FUNCTION_BLOCK  CycleHandleFB 
VAR_IN_OUT

END_VAR

VAR_INPUT
	//pFlowID: 			POINTER TO DINT :=ADR(DummyFlowID) ;
	SetEvent:			BOOL;
		
END_VAR
VAR_OUTPUT
	//Error 				: Error_Handler_typ;
END_VAR
VAR 
	// ErrorReportStruct 	:  FailureReport_Typ;	

	CMD					: Basic_cycle_CMD_typ ;
	Monitoring			: Basic_cycle_Mon_typ ;
	Status				: Basic_cycle_Status_typ ;
	Parameter			: Basic_cycle_Param_typ ;
	AtReady				: BOOL;
	Delay 				: TON ;
	StepOneShotTrig		: BOOL;
	LogMsg_0 			: LogMsg ;
	//fbClearFaultHandler_0 : fbClearFaultHandler;
	ResetError 			: R_TRIG;
	rTrigCycleDone 		: R_TRIG;
	fTrigCycleRunning 	: F_TRIG;
	rTrigCycleStart		: R_TRIG;	
	Init_trig 			: R_TRIG;
	ResetFaultTrig 		: R_TRIG;
	ResetAllTrig 		: R_TRIG;
	ResumeAllTrig 		: R_TRIG;
	LastStepMessage 	: STRING[100];
	LastStepNo 			: DINT;
	LastSubStepNo		: DINT ;
	TimeOutFault		: BOOL;
	CycleTIME 			: TON;
	StepTimerTOut 		: TON;
	SubStepTimerTOut 	: TON;
	ErrorAcknowledge 	: BOOL;
	Triger1 			: Trigger ;
	Triger2 			: Trigger ;
	Triger3 			: Trigger ;
	Triger4 			: Trigger ; 
	Triger5 			: Trigger ; 

	DummyFlowID			: DINT :=0;
	//fbCHPrgmBasic 		: FB_PrgmBasic;

	//rEvent : 			REFERENCE TO EventHelper;
	//EventHeader:		EventHeader_Typ;
	//EventParameters:	EventParam_Typ;	
END_VAR

METHOD PROTECTED CH_Logic : BOOL
VAR_STAT
	EventSent: 			BOOL;
END_VAR
VAR
	stenNomForLog	: DINT;
END_VAR

	IF CMD.LogMsgInit THEN      
		CMD.LogMsgInit := FALSE ;
		fnLogMsgInit(ADR(LogMsg_0), Parameter.ThreadName, ADR(LogGlobalArray), ADR(Parameter.PosForLog));
		LogMsg_0.Enable:= 		TRUE;
		CMD.EnableStateLogging:= TRUE;
		Parameter.ExternalLogType := LOG_INFO ;
	END_IF

	// Write state name for every change of Step Message
	IF (Monitoring.StepMessage) <> (LastStepMessage) THEN
		LastStepMessage := Monitoring.StepMessage ;
		// fnLogMsg(ADR(LogMsg_0), LOG_INFO, CONCAT(CONCAT(Parameter.CHName,', State = %d, FlowID = %d '),Monitoring.StepMessage),LastStepNo,pFlowID^,0);	
		IF CMD.EnableStateLogging THEN
			IF (Parameter.StepMessageIsForNewState) THEN
				Parameter.StepMessageIsForNewState	:= FALSE;
				stenNomForLog	:= StepNo;
			ELSE
				stenNomForLog	:= LastStepNo;
			END_IF
			fnLogMsg(ADR(LogMsg_0), LOG_INFO, CONCAT(CONCAT(CONCAT(Parameter.CHName, ', '),Monitoring.StepMessage),', State = %d.'), stenNomForLog,0,0);	
		END_IF
	END_IF
	
	

				
	//Update Step Num for Visu
	IF Triger1.EDGEPOS(Monitoring.LastStep <> Monitoring.StepNo) THEN 
		Monitoring.Visu_StepNo := LastStepNo ;
	ELSIF Status.CycleStuck AND NOT CMD.Pause THEN
		Monitoring.Visu_StepNo := Monitoring.StepNo ;
	ELSIF (Monitoring.StepNo = 0)THEN
		Monitoring.Visu_StepNo := 0 ;
	END_IF
	
	
	rTrigCycleStart(CLK:= CMD.Start);	
	IF rTrigCycleStart.Q AND Status.Running AND Monitoring.StepNo > 0 THEN
		CMD.Start:=	FALSE;		
		fnLogMsg(ADR(LogMsg_0), LOG_ERROR, CONCAT(Parameter.CHName ,' ,Start Command While Cycle Running was ignored, FlowID = %d'),0,0,0);
	END_IF

	
	(*************************** Step By Step *****************************************)
	// Step By Step Logic: If Step By Step bit set:
	//							- We stay at the same step 
	//							- We set the Pause flag
	//							- We whait for Resume bit to set to continue
	(********************************************************************)
	IF CMD.StepByStep AND (CMD.Resume OR ResumeAllTrig.Q) THEN
		CMD.Resume	:=FALSE;
		CMD.Pause	:=FALSE;
	END_IF

	IF (CMD.StepByStep AND LastStepNo <> Monitoring.StepNo)THEN
		CMD.Pause	:=TRUE;
	END_IF

	rTrigCycleDone(CLK := Status.Done);
	IF CMD.StepByStep AND rTrigCycleDone.Q THEN
		CMD.Pause	:=FALSE;
	END_IF

	(*************************** Step Time Out *****************************************)
	// Time Out Logic: If timeout elapsed:
	//							- We set the FAULT flag
	//							- We set the Error_Number and Error_Text
	//							- We set the Pause flag
	(********************************************************************)
	
	//SubStep Stuck
	Status.SubStepStuck :=  (Monitoring.SubStepNo = LastSubStepNo) AND (Status.Running) AND (Monitoring.SubStepNo <> 0);
	LastSubStepNo := Monitoring.SubStepNo;
	
	SubStepTimerTOut.PT := Parameter.TimeOut ;
	SubStepTimerTOut.IN := Status.SubStepStuck
							AND NOT CMD.Pause
							AND NOT CMD.DeactivateStepTimeOut ;
					
	SubStepTimerTOut();
	Monitoring.SubStep_TimeOut := SubStepTimerTOut.ET ;

	//Step Stuck
	Status.CycleStuck:= (LastStepNo = Monitoring.StepNo)
			 AND (Status.Running) 
			 AND Monitoring.SubStepNo = 0 ;
			
	
	StepTimerTOut.PT := Parameter.TimeOut ;
	StepTimerTOut.IN := Status.CycleStuck
							AND NOT CMD.Pause
							AND NOT CMD.StepByStep
							AND NOT CMD.DeactivateStepTimeOut ;					
	StepTimerTOut();

	Monitoring.Step_TimeOut := StepTimerTOut.ET ;
	
	
	IF StepTimerTOut.Q OR SubStepTimerTOut.Q OR SetEvent THEN
		SetEvent := FALSE ;
		Status.Fault:=	TRUE;
		TimeOutFault:=	TRUE;
	END_IF
	
		 
	IF Status.Fault THEN
		CMD.Pause := TRUE;
	END_IF

	// Logging & Event
	IF Triger2.EDGEPOS(Status.Fault) THEN
		IF TimeOutFault THEN
			IF 	Monitoring.Error_Text = Monitoring.StepMessage THEN
				fnLogMsg(ADR(LogMsg_0),
				 LOG_ERROR,
					CONCAT(
						CONCAT(
							CONCAT(Parameter.CHName,', State = %d ,SubState = %d, FlowID = %d,'),
																					Monitoring.Error_Text),
																					' ,Fault - Time Out Elaspsed'),
																						Monitoring.StepNo,
																						Monitoring.SubStepNo,0);
			ELSE
				fnLogMsg(ADR(LogMsg_0),
				 LOG_ERROR,
					CONCAT(
						CONCAT(
							CONCAT(Parameter.CHName,', State = %d ,SubState = %d, FlowID = %d,'),
																					Monitoring.Error_Text),
																					' Fault - By Event'),
																						Monitoring.StepNo,
																						Monitoring.SubStepNo,0);
			END_IF	

		//	IF NOT __ISVALIDREF(rEvent) THEN
		//		//rEvent REF=	ev_PLC_INTERNAL_TIMEOUT;	
		//		Monitoring.ExternalLogText := 'No Link to Event, send default PLC internal Timeout event';
		//		CMD.WriteExternalFaultLogCMD := TRUE;
		//	END_IF
			//fbCHPrgmBasic.mEventThrow(rEvent,ADR(EventHeader),ADR(EventParameters));
				
		ELSE
			
			fnLogMsg(ADR(LogMsg_0),
			 LOG_ERROR,
				CONCAT(
					CONCAT(
						CONCAT(Parameter.CHName,', State = %d ,SubState = %d, FlowID = %d ,'),
																				Monitoring.Error_Text),
																				' Fault - By External Event'),
																					Monitoring.StepNo,
																					Monitoring.SubStepNo,0);
		
			//Event Parames reset
			//memset(ADR(EventParameters),0,SIZEOF(EventParameters)) ;
		END_IF
		
		
	END_IF
	
	IF CMD.WriteExternalFaultLogCMD THEN
		CMD.WriteExternalFaultLogCMD := FALSE ;
		fnLogMsg(ADR(LogMsg_0), LOG_INFO, CONCAT(CONCAT(Parameter.CHName , Monitoring.ExternalLogText), ', ERROR ID = %d, FlowID = %d.'),Monitoring.ExternalLogParam1,0,0);
	END_IF
	
	IF CMD.WriteExternalLogCMD THEN
		CMD.WriteExternalLogCMD := FALSE ;
		//fnLogMsg(ADR(LogMsg_0), Parameter.ExternalLogType, CONCAT(CONCAT(Parameter.CHName,', '), Monitoring.ExternalLogText),0,0,0);
		fnLogMsg(ADR(LogMsg_0), Parameter.ExternalLogType, CONCAT(CONCAT(CONCAT(Parameter.CHName, ', ') , Monitoring.ExternalLogText), ' %d '),Monitoring.ExternalLogParam1,0,0);
	END_IF
	
	
	//StepOneShotTrig	- After Fault Handling
	IF (Monitoring.StepNo <> LastStepNo) THEN
		PrevStepNo := LastStepNo;
		LastStepNo := Monitoring.StepNo ;
		Monitoring.LastStep:= LastStepNo;
		StepOneShotTrig:=	TRUE;
		Monitoring.SubStepNo:=	0;
		//rEvent REF=	ev_PLC_INTERNAL_TIMEOUT;	
	ELSE
		StepOneShotTrig:=	FALSE;
	END_IF
	
	
	
	(*************************** Reset All *****************************************)
	// Reset All: If ResetCycle^ CMD Executed:
	//							- We reset the FAULT flag
	//							- We reset the Error_Number and Error_Text
	//							- We reset the Pause flag
	//							- We reset the Cycle^Stuck flag
	//							- We reset the Running flag
	//							- We reset the Done flag
	//							- We reset the StepNo 
	//							- We reset the StepMessage
	//							- We reset the StepByStep flag
	//							- We reset the NoFaultStep flag
	//							- We reset the ResetCycle^ flag
	//							- We reset the Delay Timer
	//							- We reset the Cycle^TimeOut_Fault flag
	(********************************************************************)	
	

	IF CMD.ResetCycle THEN
//		fnLogMsg(ADR(LogMsg_0), LOG_INFO, CONCAT(CONCAT(Parameter.CHName,', State = %d, FlowID = %d '),'Reset Cycle'),Monitoring.StepNo,pFlowID^,0);
		fnLogMsg(ADR(LogMsg_0), LOG_INFO, CONCAT(CONCAT(Parameter.CHName,', Reset Cycle, '),'State = %d.'),Monitoring.StepNo,0,0);
		Status.Fault 					:= FALSE;
		TimeOutFault					:= FALSE;
		Status.CycleStuck 				:= FALSE;
		CMD.Start 						:= FALSE;
		Status.Running 					:= FALSE;
		Status.Done 					:= FALSE;
		CMD.Pause 						:= FALSE;
		Monitoring.StepNo 				:= 0;
		Monitoring.PrevStepNo 			:= 0;
		Monitoring.SubStepNo 			:= 0;
		Monitoring.StepMessage 			:= '';
		CMD.StepByStep 					:= FALSE;
		CMD.DeactivateStepTimeOut 		:= FALSE;
		CMD.ResetCycle 					:= FALSE;
		Monitoring.Error_Text 			:= '' ;
		Monitoring.External_Error_Text 	:= '' ;
		Monitoring.ExternalLogText		:= '' ;
		Delay.IN 						:= FALSE ;
		Delay();
		Status.CycleTimeOut_Fault 		:= FALSE ;
		LastStepNo 						:= 0 ;
		LastStepMessage 				:= '';			
	END_IF
	
	
	(*************************** Resume the Cycle^ from last step ***************************)
	// Resume Logic: If No Fault and Resume bit set:
	//							- We reset the Cycle^Stuck flag
	//							- We reset the Resume
	//							- We reset the Pause flag
	(********************************************************************)
	IF NOT Status.Fault AND CMD.Resume THEN
		fnLogMsg(ADR(LogMsg_0), LOG_INFO, CONCAT(CONCAT(Parameter.CHName,', Resume, '),'State = %d.'),Monitoring.StepNo,0,0);
//		fnLogMsg(ADR(LogMsg_0), LOG_INFO, CONCAT(CONCAT(Parameter.CHName,', State = %d, FlowID = %d '),'Resume'),Monitoring.StepNo,pFlowID^,0);
		CMD.Pause 			:= FALSE;
		Status.CycleStuck 	:= FALSE;
		CMD.Resume 			:= FALSE;
		StepOneShotTrig		:= TRUE;
	END_IF

	
	(*************************** Auto Errors Reset ***************************)
	// Errors Logic: If No Fault and not Cycle^TimeOut_Fault:
	//							- We reset the Error_Num 
	//							- We reset the Error_Text
	(********************************************************************)
	IF NOT Status.Fault AND NOT Status.CycleTimeOut_Fault THEN
		Monitoring.Error_Text 			:= '' ;
		Monitoring.External_Error_Text 	:= '' ;
	END_IF
	
	
	(*************************** Errors Reset ***************************)
	// Errors Logic: If ResetErr bit set:
	//							- We reset the Error_Num 
	//							- We reset the Error_Text
	//							- We reset the Pause flag
	//							- We reset the Fault flag
	//							- We reset the Cycle^TimeOut_Fault flag
	(********************************************************************)
	//ResetFaultTrig.CLK := CMD.ResetErr ;
	//ResetFaultTrig();
	IF (*ResetFaultTrig.Q*)CMD.ResetErr THEN
		CMD.ResetErr := FALSE ;
		fnLogMsg(ADR(LogMsg_0), LOG_INFO, CONCAT(CONCAT(Parameter.CHName,', Reset Error, '),'State = %d, FlowID = %d.'),Monitoring.StepNo,0,0);
		Monitoring.Error_Text 			:= '' ;
		Monitoring.External_Error_Text 	:= '' ;
		
		Status.Fault 					:= FALSE ;
		TimeOutFault					:= FALSE ;
		Status.CycleTimeOut_Fault 		:= FALSE ;
	END_IF
	
	
	//Cycle^ TIME
	IF CMD.Deacivate_Sequence_Time_Out = FALSE THEN
		(*************************** Monitoring Last Cycle^ Time ***************************)
		// Last Cycle^ Time Logic: If Running flag bit set:
		//						  - We set the LastCycle^Time to Cycle^Time.ET
		(********************************************************************)
		fTrigCycleRunning.CLK			:= Status.Running ;
		fTrigCycleRunning();
		IF fTrigCycleRunning.Q THEN
			Monitoring.LastCycleTIME 	:= CycleTIME.ET;
		END_IF
	
 
		(*************************** Seting the tiem of Cycle^ Time Out ***************************)
		// Cycle^ Time Out Logic: If Cycle^TimeOut > 0:
		//						  - We set the Cycle^Time.PT to Cycle^TimeOut
		(********************************************************************)
		IF TIME_TO_DINT(Parameter.CycleTimeOut) > 0 THEN
			CycleTIME.PT := (Parameter.CycleTimeOut) ;
		ELSE
			CycleTIME.PT := T#30M ;
		END_IF
		
		(*************************** Cycle^ Time set ***************************)
		// Cycle^ Time set Logic: If Running and not Cycle^TimeOut_Fault and not Deacivate_Sequence_Time_Out :
		//						  - We set the Cycle^Time.IN 
		(********************************************************************)
		CycleTIME.IN := Status.Running AND NOT Status.CycleTimeOut_Fault (*AND NOT CMD.Deacivate_Sequence_Time_Out *);
		CycleTIME();
		
		
		(*************************** Cycle^ Time Out ***************************)
		// Cycle^ Time Out Logic: If Cycle^Time.Q bit set:
		//							- We set the Error_Text
		//							- We set the Pause flag
		//							- We set the Cycle^TimeOut_Fault flag
		(********************************************************************)
		IF CycleTIME.Q THEN
			CMD.Pause 					:= TRUE ;
			Status.CycleTimeOut_Fault 	:= TRUE ;
			Monitoring.Error_Text 		:= 'Sequence Time Out' ;
		END_IF
		
		Monitoring.CycleTIME 	:= CycleTIME.ET ;
	END_IF
	

	

	
	//fbCHPrgmBasic();

	//fnLogTransfer FUNCTION call
	fnLogTransfer(ADR(LogMsg_0));
END_METHOD

PROPERTY PUBLIC CHName : STRING
GET
CHName := THIS^.Parameter.CHName ;
END_GET
SET
THIS^.Parameter.CHName := CHName ;
END_SET
END_PROPERTY

PROPERTY PUBLIC CycleTimeOut : TIME
GET
CycleTimeOut := THIS^.Parameter.CycleTimeOut ;
END_GET
SET
THIS^.Parameter.CycleTimeOut := CycleTimeOut ;
END_SET
END_PROPERTY

PROPERTY PUBLIC Deacivate_Sequence_Time_Out : BOOL
GET
Deacivate_Sequence_Time_Out := THIS^.CMD.Deacivate_Sequence_Time_Out ;
END_GET
SET
THIS^.CMD.Deacivate_Sequence_Time_Out := Deacivate_Sequence_Time_Out ;
END_SET
END_PROPERTY

PROPERTY PUBLIC DeactivateStepTimeOut : BOOL
GET
DeactivateStepTimeOut := THIS^.CMD.DeactivateStepTimeOut ;
END_GET
SET
THIS^.CMD.DeactivateStepTimeOut := DeactivateStepTimeOut ;
END_SET
END_PROPERTY

PROPERTY PUBLIC Done : BOOL
GET
Done := THIS^.Status.Done ;
END_GET
END_PROPERTY

PROPERTY PUBLIC Error_Text : STRING
GET
Error_Text := THIS^.Monitoring.Error_Text ;
END_GET
SET // PUBLIC
THIS^.Monitoring.Error_Text := Error_Text;
END_SET
END_PROPERTY

PROPERTY PUBLIC ExternalLogParam1 : DINT
GET
ExternalLogParam1 := THIS^.Monitoring.ExternalLogParam1;
END_GET
SET
THIS^.Monitoring.ExternalLogParam1 := ExternalLogParam1;
END_SET
END_PROPERTY

PROPERTY PUBLIC ExternalLogText : STRING
GET
ExternalLogText := THIS^.Monitoring.ExternalLogText ;
END_GET
SET
THIS^.Monitoring.ExternalLogText := ExternalLogText ;
END_SET
END_PROPERTY

PROPERTY PUBLIC Fault : BOOL
GET
Fault := THIS^.Status.Fault ;
END_GET
SET
THIS^.Status.Fault := Fault ;
END_SET
END_PROPERTY

PROPERTY PUBLIC LogEnable : BOOL
SET
CMD.EnableStateLogging:= LogEnable ;
END_SET
END_PROPERTY

PROPERTY PUBLIC Pause : BOOL
GET

	Pause := THIS^.CMD.Pause ;
END_GET
SET
 
	THIS^.CMD.Pause := Pause ;
END_SET
END_PROPERTY

PROPERTY PUBLIC pLogMsg_0 : POINTER TO LogMsg
GET
pLogMsg_0:= ADR(THIS^.LogMsg_0);
END_GET
END_PROPERTY

PROPERTY PUBLIC PosForLog : USINT
SET
THIS^.Parameter.PosForLog := PosForLog ;
END_SET
END_PROPERTY

PROPERTY PUBLIC PrevStepNo : DINT
GET
PrevStepNo := THIS^.Monitoring.PrevStepNo ;
END_GET
SET
THIS^.Monitoring.PrevStepNo := PrevStepNo;
END_SET
END_PROPERTY

PROPERTY PUBLIC ResetCycle : BOOL
SET

THIS^.CMD.ResetCycle := ResetCycle ;
END_SET
END_PROPERTY

PROPERTY PUBLIC ResetErr : BOOL
SET
THIS^.CMD.ResetErr := ResetErr ;
END_SET
END_PROPERTY

PROPERTY PUBLIC Resume : BOOL
SET
THIS^.CMD.Resume := Resume ;
END_SET
END_PROPERTY

PROPERTY PUBLIC Running : BOOL
GET
Running := This^.Status.Running ;
END_GET
END_PROPERTY

METHOD SetStepNoWithName
VAR_INPUT
	stepNpmber : DINT;
END_VAR
VAR_IN_OUT
	stateNames : ARRAY [*] OF STRING(32); // in only
END_VAR
StepNo										:= stepNpmber;
Parameter.StepMessageIsForNewState	:= TRUE;;
IF (stepNpmber >= LOWER_BOUND(stateNames,1) AND stepNpmber <= UPPER_BOUND(stateNames,1)) THEN
	Monitoring.StepMessage			:= stateNames[stepNpmber];
ELSE
	Monitoring.StepMessage			:= 'NO_Name_Step';
END_IF
END_METHOD

PROPERTY PUBLIC Start : BOOL
GET

Start := THIS^.CMD.Start ;
END_GET
SET

 THIS^.CMD.Start := Start ;
END_SET
END_PROPERTY

PROPERTY PUBLIC StepByStep : BOOL
GET

StepByStep := THIS^.CMD.StepByStep ;
END_GET
SET
THIS^.CMD.StepByStep := StepByStep ;
END_SET
END_PROPERTY

PROPERTY PUBLIC StepMessage : STRING
GET
StepMessage := THIS^.Monitoring.StepMessage ;
END_GET
SET
THIS^.Monitoring.StepMessage := StepMessage ;
END_SET
END_PROPERTY

PROPERTY PUBLIC StepNo : DINT
GET
StepNo := THIS^.Monitoring.StepNo ;
END_GET
SET
THIS^.Monitoring.StepNo := StepNo ;
END_SET
END_PROPERTY

PROPERTY PUBLIC StepStuck : BOOL
GET
StepStuck := THIS^.Status.CycleStuck;
END_GET
END_PROPERTY

PROPERTY SubStepNo : DINT
GET
SubStepNo := THIS^.Monitoring.SubStepNo ;
END_GET
SET
THIS^.Monitoring.SubStepNo := SubStepNo ;
END_SET
END_PROPERTY

PROPERTY PUBLIC SubStepStuck : BOOL
GET
SubStepStuck := THIS^.Status.SubStepStuck;
END_GET
END_PROPERTY

PROPERTY PUBLIC ThreadName : STRING
GET
ThreadName := THIS^.Parameter.ThreadName ;
END_GET
SET
THIS^.Parameter.ThreadName := ThreadName ;
END_SET
END_PROPERTY

PROPERTY PUBLIC TimeOut : TIME
GET
TimeOut := THIS^.Parameter.TimeOut ;
END_GET
SET
THIS^.Parameter.TimeOut := TimeOut ;
END_SET
END_PROPERTY

PROPERTY WriteExternalFaultLog : BOOL
SET
 THIS^.CMD.WriteExternalFaultLogCMD := WriteExternalFaultLog ;
END_SET
END_PROPERTY

PROPERTY WriteExternalLog : BOOL
GET
WriteExternalLog:= THIS^.CMD.WriteExternalLogCMD;
END_GET
SET
 THIS^.CMD.WriteExternalLogCMD := WriteExternalLog ;
END_SET
END_PROPERTY

END_FUNCTION_BLOCK

(* stored: Version 1.1.0.1, ProductVersion 3.1.4024.3
   POU CycleHandleFB: Id {7735e37c-79e6-0564-0a01-368493b6cfae}, SpecialFunc None
   Method CH_Logic: Id {de92f3d3-5eef-08e7-150f-1053c8bfc5d4}
   Property CHName: Id {b719a3a9-b74c-0611-00c1-938ab447f405}
   Get Get: Id {c8a0b1a7-83df-0c4b-1b7a-039ce570bce4}
   Set Set: Id {8e67b140-033d-0515-33d0-83db229bfb63}
   Property CycleTimeOut: Id {7d0818f7-785b-0dec-13c2-436c3d3645af}
   Get Get: Id {6022127a-85c7-0a3e-3a10-07376c59ef3e}
   Set Set: Id {549b9d83-033d-0411-11ea-d22fe550ca6d}
   Property Deacivate_Sequence_Time_Out: Id {5d479b4e-525f-0c04-035e-90afffcbd973}
   Get Get: Id {e100964d-ce50-0fcf-1494-78ab87dd5eaa}
   Set Set: Id {a79f8032-492f-0fad-1119-966147d3d705}
   Property DeactivateStepTimeOut: Id {129c3ab4-2e95-08e9-2f57-3712c9787463}
   Get Get: Id {40625825-15f6-0f44-0106-3ea73bf4d5c9}
   Set Set: Id {3a102886-0984-053e-38eb-8d6ea88337f0}
   Property Done: Id {d1e3a8ce-4706-0eda-234e-9cf57ecb3869}
   Get Get: Id {5b88c89d-9965-0ffc-3e44-30aa6c81d06c}
   Property Error_Text: Id {84a8b9c2-522e-0958-01b4-9461a3d3ff96}
   Get Get: Id {b7615acb-012c-001a-0fee-d344c12db797}
   Set Set: Id {544018e2-1e01-4f7f-b317-cc769c88eccd}
   Property ExternalLogParam1: Id {941372f5-4df1-039c-12d9-48b506e51c1b}
   Get Get: Id {589b08d3-1c39-00a4-01b5-a9bdee876480}
   Set Set: Id {808722a1-3bec-0b9b-26d2-a0a03e6dc3e3}
   Property ExternalLogText: Id {fc8da912-f436-03c7-052a-f14450f8a0f2}
   Get Get: Id {594302de-67b2-0087-00cb-3c10e477cf3e}
   Set Set: Id {039ad526-1940-0528-1e20-ca1f00114d77}
   Property Fault: Id {4af4f8c6-56ed-05f4-100e-0be7218b0616}
   Get Get: Id {0ab5679e-0626-0a55-1eca-25d7e5f27d10}
   Set Set: Id {8ebc7d74-b6e0-01f6-15e4-f98805c451de}
   Property LogEnable: Id {a4e681b8-8b20-0429-3d73-b8e81565a348}
   Set Set: Id {75f8e8eb-6198-09a5-2e84-43b41e5a8593}
   Property Pause: Id {2b88fb58-9da8-038f-15e5-45bc113046a7}
   Get Get: Id {a89518c4-761b-0f3f-345f-692561305275}
   Set Set: Id {fd95c578-29b7-0191-0483-43de6af40021}
   Property pLogMsg_0: Id {06b13c61-cf02-002c-0b6f-a8f7305203f4}
   Get Get: Id {292facf3-b74e-0762-20ac-b39a05b226af}
   Property PosForLog: Id {127d07e4-cbef-0d00-1fe2-0ff5f5fa06bc}
   Set Set: Id {672f4656-2c56-0f63-3569-5bbabfa2a5c0}
   Property PrevStepNo: Id {e4f63e9d-7718-034a-2a4a-6f3c98a63f78}
   Get Get: Id {1f1dd22e-f678-0725-0924-3e6606439645}
   Set Set: Id {73d89c05-5038-08a0-0de8-328b2f6eb23f}
   Property ResetCycle: Id {29fa3b2e-271f-06ef-2071-79685869cf26}
   Set Set: Id {03c8adcb-4411-0e78-3a2a-3cc454357c0d}
   Property ResetErr: Id {e59909a5-de76-0166-3d50-c57abf060429}
   Set Set: Id {25f2259c-72c2-0507-0cd7-82f31553f111}
   Property Resume: Id {45bf2488-2a88-0ccd-284b-d3058b659911}
   Set Set: Id {136479fc-717f-0cad-3ad0-f015b0a0fa1e}
   Property Running: Id {734192bc-411a-022c-309d-0ac43d9307cf}
   Get Get: Id {ce8f832e-c538-0aae-1b0f-d9aa7983218a}
   Method SetStepNoWithName: Id {f884aca0-9f99-4e2a-ac39-e11e61111c8c}
   Property Start: Id {6db37d9c-9cb9-0c3e-09dd-eebcbf691404}
   Get Get: Id {7477e5bf-5e80-08c8-03d6-feb13b85c5e2}
   Set Set: Id {1e795450-f44d-05b4-3e9a-735e20fa9574}
   Property StepByStep: Id {5adf3970-e29f-0b79-25d9-cdea137534dd}
   Get Get: Id {2919a340-049c-0c81-2235-247ec8cf5edb}
   Set Set: Id {b40835a8-bb94-03bf-37ef-9f35ede9eaa0}
   Property StepMessage: Id {5b0aec22-e6e0-0c02-31f3-d4b10459704c}
   Get Get: Id {3ed7f2c1-a1ae-0536-0ebd-e2947c4dc3e5}
   Set Set: Id {bdbfa284-680a-0851-1ec0-c5745ce9beb9}
   Property StepNo: Id {9a0097f5-4123-0fbd-0e5f-701b97b95848}
   Get Get: Id {636d5f47-f4a2-084f-18a6-e56171e7afde}
   Set Set: Id {af18b08e-4470-08f3-3295-d9603a7219cb}
   Property StepStuck: Id {237b46fb-1e91-0ab5-2a91-f28da83c451d}
   Get Get: Id {53d6adf3-86b3-08e8-2b3c-042f4993335a}
   Property SubStepNo: Id {9c9f1aa8-d3a9-0d82-38cd-53dfed62153b}
   Get Get: Id {3a4d00fc-7329-0fc8-0b71-4cff685464d0}
   Set Set: Id {9db73600-b841-00f8-20a2-605dbfa4927c}
   Property SubStepStuck: Id {c3c6267b-2a5b-0ff0-1f88-dff9850d9a65}
   Get Get: Id {66007776-a817-0c56-28ad-0e3be4506a31}
   Property ThreadName: Id {3aff06ef-83d0-0000-38f3-c0ec53c44951}
   Get Get: Id {015c9453-2c49-0f3e-1db8-ddb183617302}
   Set Set: Id {b58a3ae3-305d-098d-3548-d19139750819}
   Property TimeOut: Id {0d6ded26-6e47-08b7-29cb-f943c84136c4}
   Get Get: Id {198a6246-3940-0943-01e0-a8dfe98c33ec}
   Set Set: Id {c1314f8c-e4f3-061f-0a5b-822e3a456917}
   Property WriteExternalFaultLog: Id {f55e0386-0396-025c-14db-18a3e3ef98fc}
   Set Set: Id {f684ac2f-66f0-00e6-0e27-202f6aa28988}
   Property WriteExternalLog: Id {9b551ea8-4243-02bf-2e7a-5b1e08ac80d7}
   Get Get: Id {b019b58a-9a0a-06c0-3fc7-687741b8dec4}
   Set Set: Id {5c151df8-0089-0518-0f12-c1c2c88ffa86} *)
